// Mitsubishi GX Works2 project: 0625(점멸회로_무한루프)   PLC: Q02/Q02H

PROGRAM MAIN
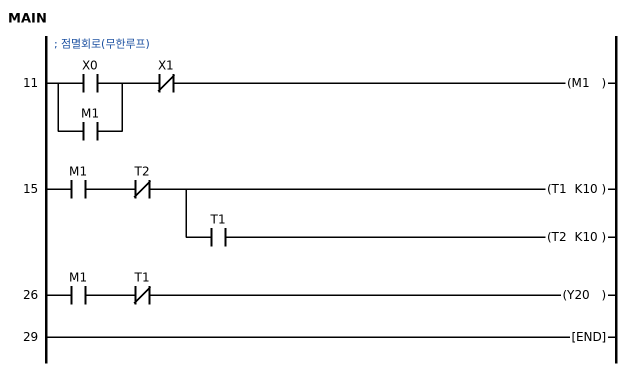
; 점멸회로(무한루프)
11    LD      X0
      OR      M1
      ANI     X1
      OUT     M1
15    LD      M1
      ANI     T2
      OUT     T1 K10
      AND     T1
      OUT     T2 K10
26    LD      M1
      ANI     T1
      OUT     Y20
29    END
END_PROGRAM
